FUNCTION_BLOCK ABSTRACT FB_Handler IMPLEMENTS I_Handler
VAR_INPUT
END_VAR
VAR_OUTPUT
END_VAR
VAR
	iNextHandler:			I_Handler;
END_VAR

//	The FB_Handler is an abstract function block that implements the I_Handler interface. 
//	It represents a handler in the Chain of Responsibility pattern,
//	where a request can be passed along a chain of potential handlers until one of them handles the request.
//	Each handler in the chain has the ability to either handle the request or pass it to the next handle

METHOD PUBLIC M_Request
VAR_INPUT
	stEvent:			ST_Event;		// event to be handled. 
END_VAR
// The M_Request method is used to handle the request.

IF iNextHandler <> 0 THEN
	// the request is passed to the next handler 
	iNextHandler.M_Request(stEvent);
END_IF
END_METHOD

METHOD PUBLIC M_SetNext
VAR_INPUT
	iHandler:				I_Handler;
END_VAR
// next handler in the chain
iNextHandler:= iHandler;
END_METHOD

END_FUNCTION_BLOCK

(* stored: Version 1.1.0.1, ProductVersion 3.1.4024.12
   POU FB_Handler: Id {5b555d9d-9f1a-4168-ace2-3a53af448bf3}, SpecialFunc None
   Method M_Request: Id {0dbdffe3-6983-4b80-bcf0-f4c7d261385e}
   Method M_SetNext: Id {2277a74c-b100-4336-aa47-a0aa9f65da8c} *)
